Fanuc KAREL source: kb00009.KL

-- PROVISIONAL review KL for V1013-1; original PC SHA256 61aaf5b12ca823cf904656eb97254ab24226acdf3383ab3cde1a8b56c524cfde
-- Incomplete behavior may be omitted. Consult companion uncertainty JSON. Do not deploy.
PROGRAM KB00009
%NOLOCKGROUP
VAR
  P1 : REAL
  P2 : REAL
  RESULT : REAL
BEGIN
  -- UNRESOLVED_PC offsets 5-16; opcodes 2E,23
  -- UNRESOLVED_PC offsets 21-32; opcodes 2E,23
  -- UNRESOLVED_PC offsets 37-58; opcodes 27,22,22,76,23
  -- UNRESOLVED_PC offsets 63-67; opcodes 7F
END KB00009
